{attribute 'Tc2GvlVarNames'}
VAR_GLOBAL
END_VAR

(* stored: Version 1.1.0.1, ProductVersion 3.1.4020.12
   GVL Globale_Variablen: Id {b60774ce-8525-4514-a2f7-a92e506b15c4} *)
